FUNCTION_BLOCK FeedInfluentBasic (* Basic Function Block Type *)
  (* Standard: 61499-2 *)
  (* Version 0.0, 6/13/2026, Schneider Electric, Template *)
  PACKAGE SE.Nereda;
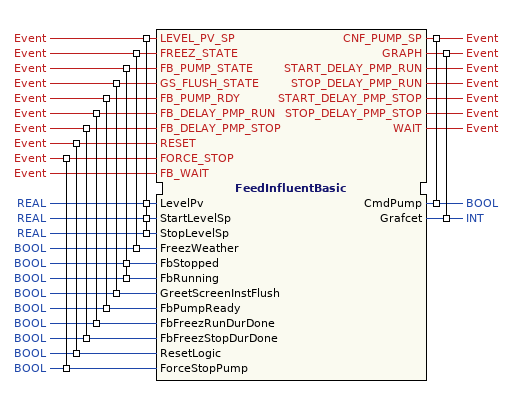
  EVENT_INPUT
    LEVEL_PV_SP WITH StartLevelSp, StopLevelSp, LevelPv;
    FREEZ_STATE WITH FreezWeather;
    FB_PUMP_STATE WITH FbStopped, FbRunning;
    GS_FLUSH_STATE WITH GreetScreenInstFlush;
    FB_PUMP_RDY WITH FbPumpReady;
    FB_DELAY_PMP_RUN WITH FbFreezRunDurDone;
    FB_DELAY_PMP_STOP WITH FbFreezStopDurDone;
    RESET WITH ResetLogic;
    FORCE_STOP WITH ForceStopPump;
    FB_WAIT;
  END_EVENT
  EVENT_OUTPUT
    CNF_PUMP_SP WITH CmdPump;
    GRAPH WITH Grafcet;
    START_DELAY_PMP_RUN;
    STOP_DELAY_PMP_RUN;
    START_DELAY_PMP_STOP;
    STOP_DELAY_PMP_STOP;
    WAIT;
  END_EVENT
  VAR_INPUT
    LevelPv : REAL;
    StartLevelSp : REAL;
    StopLevelSp : REAL;
    FreezWeather : BOOL;
    FbStopped : BOOL;
    FbRunning : BOOL;
    GreetScreenInstFlush : BOOL;
    FbPumpReady : BOOL;
    FbFreezRunDurDone : BOOL;
    FbFreezStopDurDone : BOOL;
    ResetLogic : BOOL;
    ForceStopPump : BOOL;
  END_VAR
  VAR_OUTPUT
    CmdPump : BOOL;
    Grafcet : INT;
  END_VAR
  VAR
    FreezeMode : BOOL;
  END_VAR
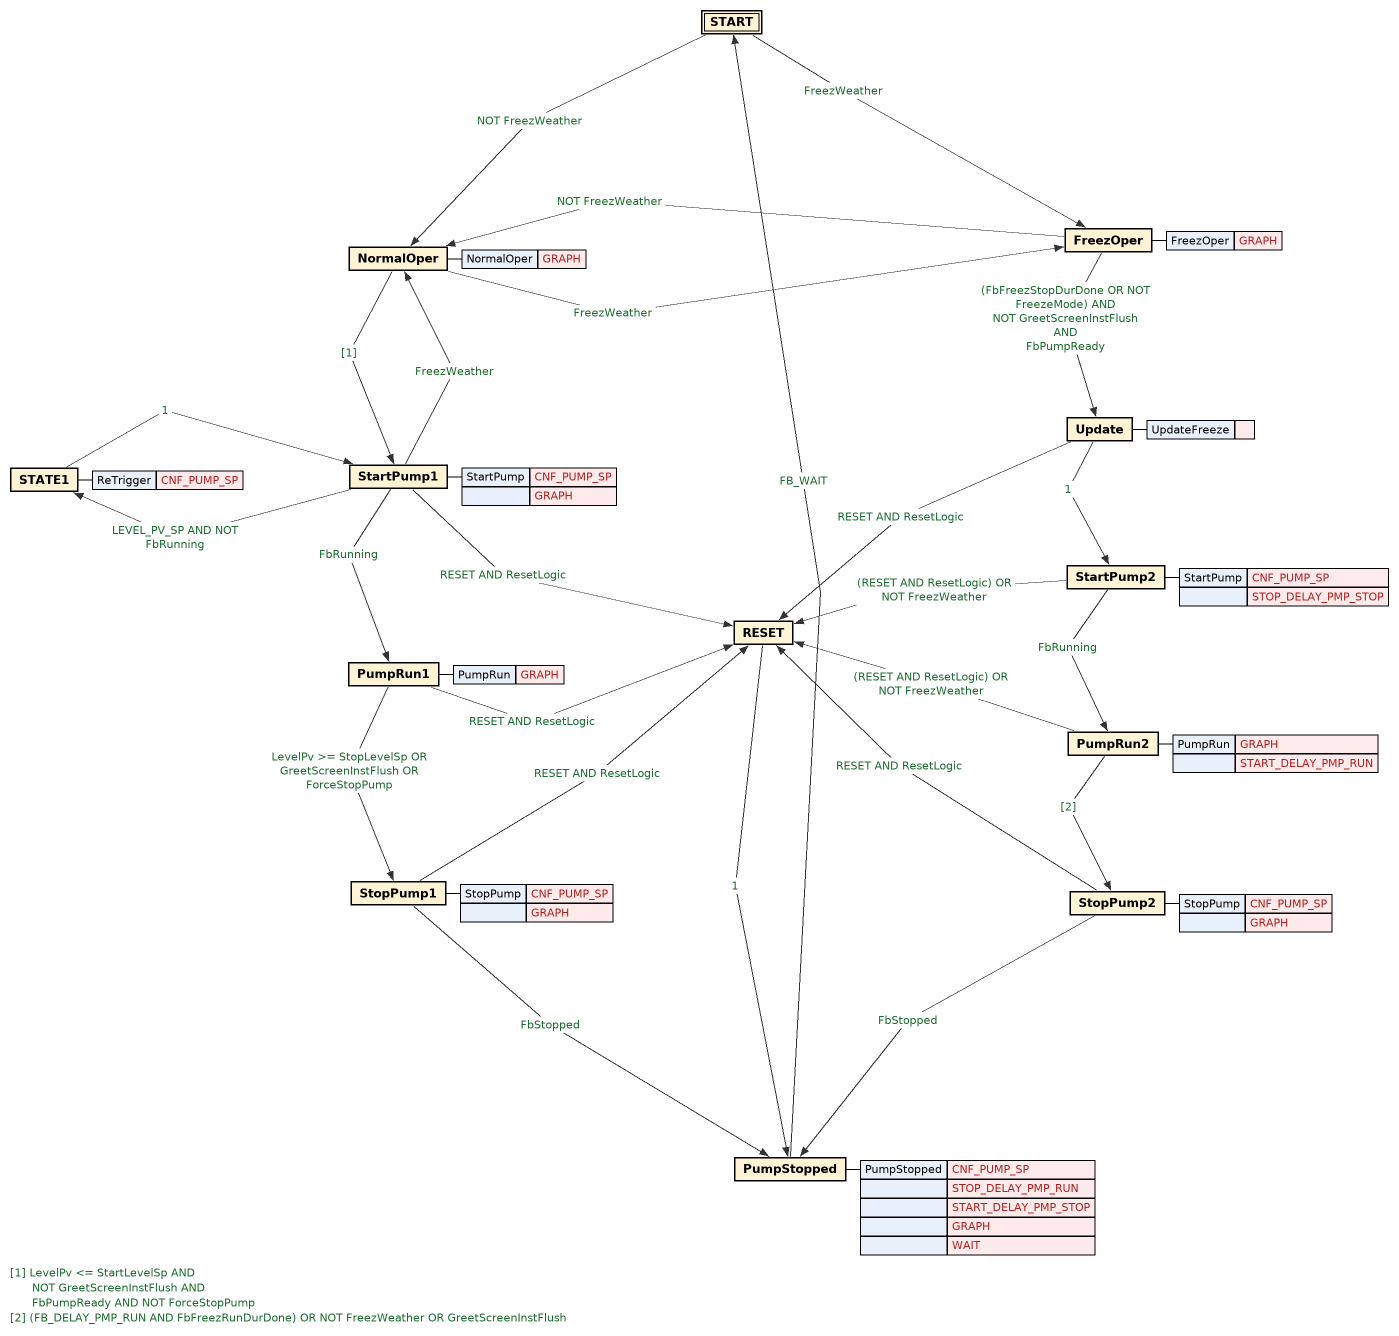
  EC_STATES
    START; (* Initial State *)
    NormalOper : NormalOper -> GRAPH;
    FreezOper : FreezOper -> GRAPH;
    StartPump1 : StartPump -> CNF_PUMP_SP, -> GRAPH;
    StopPump1 : StopPump -> CNF_PUMP_SP, -> GRAPH;
    PumpRun1 : PumpRun -> GRAPH;
    StartPump2 : StartPump -> CNF_PUMP_SP, -> STOP_DELAY_PMP_STOP;
    StopPump2 : StopPump -> CNF_PUMP_SP, -> GRAPH;
    PumpRun2 : PumpRun -> GRAPH, -> START_DELAY_PMP_RUN;
    PumpStopped : PumpStopped -> CNF_PUMP_SP, -> STOP_DELAY_PMP_RUN, -> START_DELAY_PMP_STOP, -> GRAPH, -> WAIT;
    Update : UpdateFreeze;
    RESET;
    STATE1 : ReTrigger -> CNF_PUMP_SP;
  END_STATES
  EC_TRANSITIONS
    START TO FreezOper := FreezWeather;
    START TO NormalOper := NOT FreezWeather;
    NormalOper TO FreezOper := FreezWeather;
    FreezOper TO NormalOper := NOT FreezWeather;
    NormalOper TO StartPump1 := LevelPv <= StartLevelSp AND NOT GreetScreenInstFlush AND FbPumpReady AND NOT ForceStopPump;
    PumpRun1 TO StopPump1 := LevelPv >= StopLevelSp OR GreetScreenInstFlush OR ForceStopPump;
    StopPump1 TO PumpStopped := FbStopped;
    StartPump1 TO PumpRun1 := FbRunning;
    PumpStopped TO START := FB_WAIT;
    FreezOper TO Update := (FbFreezStopDurDone OR NOT FreezeMode) AND NOT GreetScreenInstFlush AND FbPumpReady;
    StartPump2 TO PumpRun2 := FbRunning;
    PumpRun2 TO StopPump2 := (FB_DELAY_PMP_RUN AND FbFreezRunDurDone) OR NOT FreezWeather OR GreetScreenInstFlush;
    StopPump2 TO PumpStopped := FbStopped;
    Update TO StartPump2 := 1;
    StartPump1 TO RESET := RESET AND ResetLogic;
    PumpRun1 TO RESET := RESET AND ResetLogic;
    StopPump1 TO RESET := RESET AND ResetLogic;
    StopPump2 TO RESET := RESET AND ResetLogic;
    PumpRun2 TO RESET := (RESET AND ResetLogic) OR NOT FreezWeather;
    StartPump2 TO RESET := (RESET AND ResetLogic) OR NOT FreezWeather;
    Update TO RESET := RESET AND ResetLogic;
    StartPump1 TO STATE1 := LEVEL_PV_SP AND NOT FbRunning;
    StartPump1 TO NormalOper := FreezWeather;
    STATE1 TO StartPump1 := 1;
    RESET TO PumpStopped := 1;
  END_TRANSITIONS
  ALGORITHM StartPump IN ST:
;
CmdPump := TRUE;

IF Grafcet = 1 THEN
	Grafcet := 2;
ELSIF Grafcet = 10 THEN
	Grafcet := 11;
END_IF;
  END_ALGORITHM
  ALGORITHM StopPump IN ST:
;
CmdPump := FALSE;

IF Grafcet = 3 THEN
	Grafcet := 4;
ELSIF Grafcet = 12 THEN
	Grafcet := 13;
END_IF;
  END_ALGORITHM
  ALGORITHM NormalOper IN ST:
;
Grafcet := 1;
FreezeMode := FALSE;
  END_ALGORITHM
  ALGORITHM FreezOper IN ST:
;
Grafcet := 10;
  END_ALGORITHM
  ALGORITHM PumpRun IN ST:
;
IF Grafcet = 2 THEN
	Grafcet := 3;
ELSIF Grafcet = 11 THEN
	Grafcet := 12;
END_IF;
  END_ALGORITHM
  ALGORITHM PumpStopped IN ST:
;
CmdPump := FALSE;
Grafcet := 9;
  END_ALGORITHM
  ALGORITHM UpdateFreeze IN ST:
;
FreezeMode := TRUE;
  END_ALGORITHM
  ALGORITHM Reset IN ST:
;
CmdPump := FALSE;
  END_ALGORITHM
  ALGORITHM ReTrigger IN ST:
;
CmdPump := FALSE;
  END_ALGORITHM
END_FUNCTION_BLOCK
